FUNCTION_BLOCK basicNecessidade2Equipamentos (* Basic Function Block Type *)
  (* Standard: 61499-2 *)
  (* Version 0.0, 24/02/2026, Template *)
  PACKAGE Hidryco.HidrycoLib;
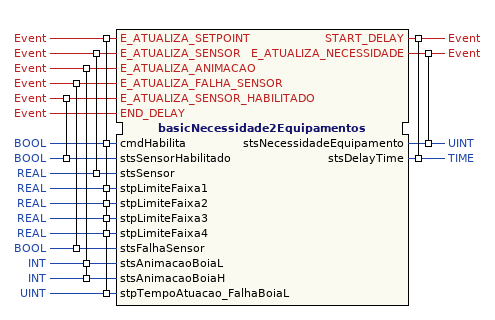
  EVENT_INPUT
    E_ATUALIZA_SETPOINT WITH stpLimiteFaixa1, stpLimiteFaixa2, stpLimiteFaixa3, stpLimiteFaixa4, stpTempoAtuacao_FalhaBoiaL, cmdHabilita;
    E_ATUALIZA_SENSOR WITH stsSensor;
    E_ATUALIZA_ANIMACAO WITH stsAnimacaoBoiaL, stsAnimacaoBoiaH;
    E_ATUALIZA_FALHA_SENSOR WITH stsFalhaSensor;
    E_ATUALIZA_SENSOR_HABILITADO WITH stsSensorHabilitado;
    END_DELAY;
  END_EVENT
  EVENT_OUTPUT
    START_DELAY WITH stsDelayTime;
    E_ATUALIZA_NECESSIDADE WITH stsNecessidadeEquipamento;
  END_EVENT
  VAR_INPUT
    cmdHabilita : BOOL;
    stsSensorHabilitado : BOOL;
    stsSensor : REAL;
    stpLimiteFaixa1 : REAL;
    stpLimiteFaixa2 : REAL;
    stpLimiteFaixa3 : REAL;
    stpLimiteFaixa4 : REAL;
    stsFalhaSensor : BOOL;
    stsAnimacaoBoiaL : INT;
    stsAnimacaoBoiaH : INT;
    stpTempoAtuacao_FalhaBoiaL : UINT; (* Tempo para equipamento ficar ligado quando bater na boia H e a boia L estiver em falha *)
  END_VAR
  VAR_OUTPUT
    stsNecessidadeEquipamento : UINT;
    stsDelayTime : TIME;
  END_VAR
  VAR
    auxiliar : INT := 0;
  END_VAR
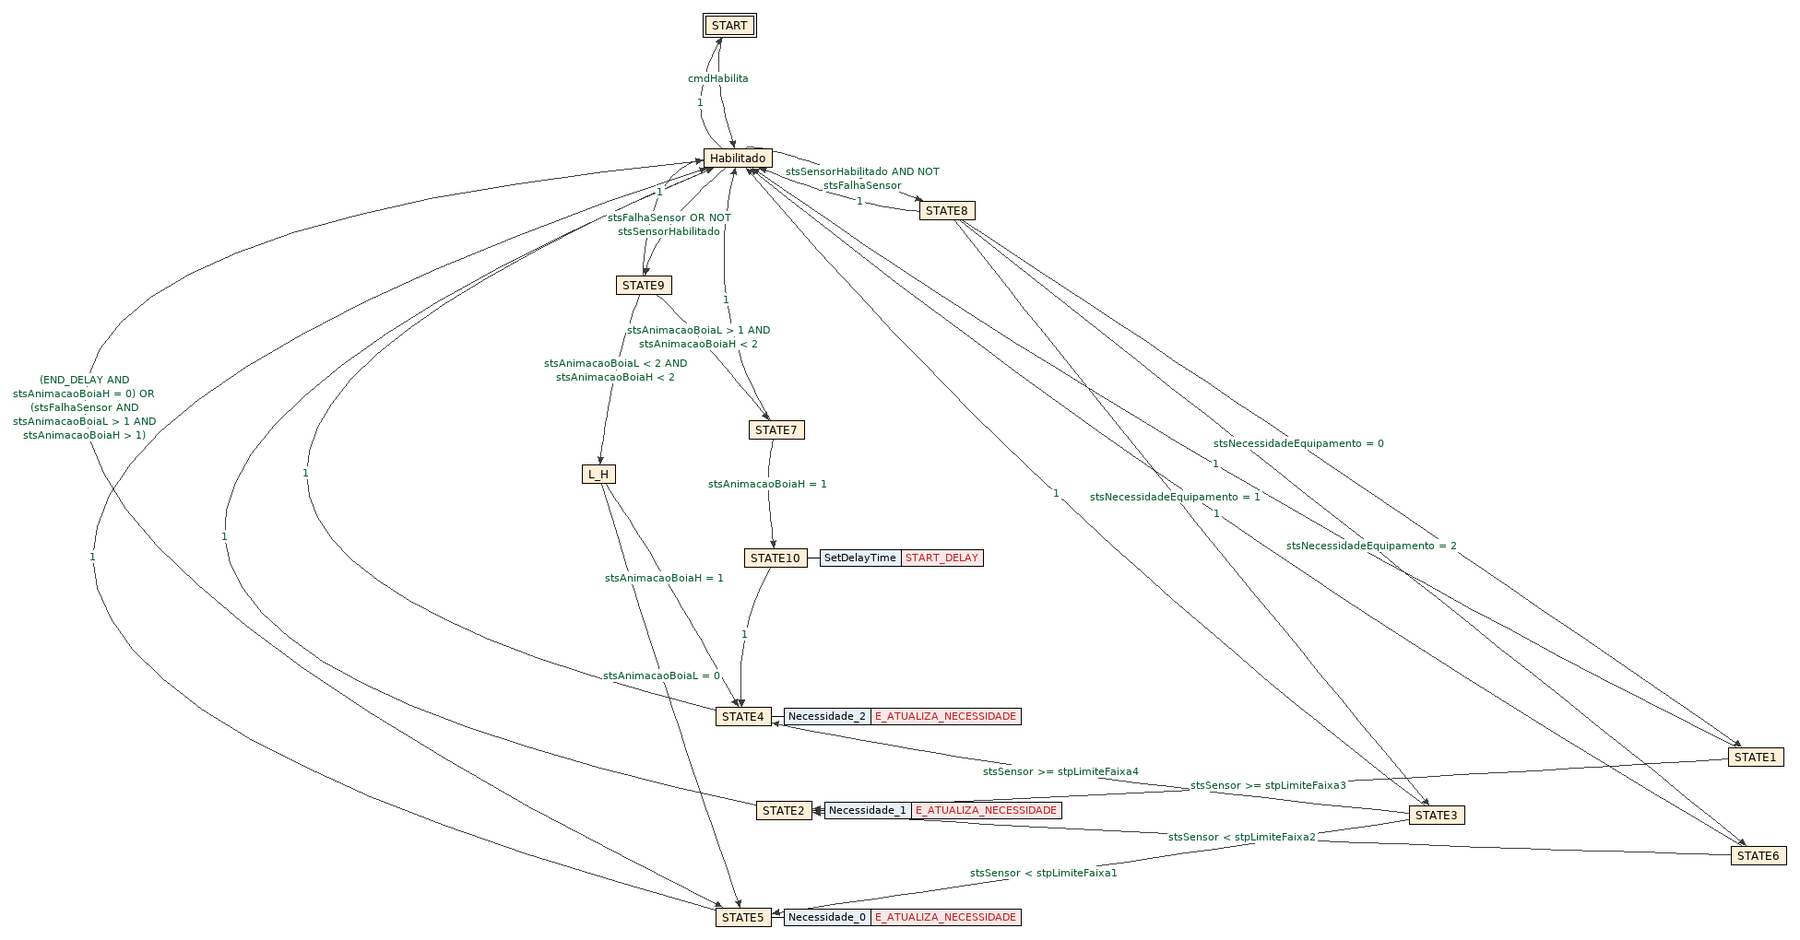
  EC_STATES
    START; (* Initial State *)
    STATE1;
    STATE2 : Necessidade_1 -> E_ATUALIZA_NECESSIDADE;
    STATE3;
    STATE4 : Necessidade_2 -> E_ATUALIZA_NECESSIDADE;
    STATE5 : Necessidade_0 -> E_ATUALIZA_NECESSIDADE;
    STATE6;
    STATE8;
    STATE9;
    L_H;
    STATE7;
    STATE10 : SetDelayTime -> START_DELAY;
    Habilitado;
  END_STATES
  EC_TRANSITIONS
    START TO Habilitado := cmdHabilita;
    Habilitado TO STATE8 := stsSensorHabilitado AND NOT stsFalhaSensor;
    STATE8 TO STATE1 := stsNecessidadeEquipamento = 0;
    STATE1 TO STATE2 := stsSensor >= stpLimiteFaixa3;
    STATE8 TO STATE3 := stsNecessidadeEquipamento = 1;
    STATE3 TO STATE4 := stsSensor >= stpLimiteFaixa4;
    STATE3 TO STATE5 := stsSensor < stpLimiteFaixa1;
    STATE8 TO STATE6 := stsNecessidadeEquipamento = 2;
    STATE6 TO STATE2 := stsSensor < stpLimiteFaixa2;
    STATE8 TO Habilitado := 1;
    Habilitado TO STATE9 := stsFalhaSensor OR NOT stsSensorHabilitado;
    STATE9 TO L_H := stsAnimacaoBoiaL < 2 AND stsAnimacaoBoiaH < 2;
    L_H TO STATE4 := stsAnimacaoBoiaH = 1;
    L_H TO STATE5 := stsAnimacaoBoiaL = 0;
    STATE9 TO STATE7 := stsAnimacaoBoiaL > 1 AND stsAnimacaoBoiaH < 2;
    STATE7 TO STATE10 := stsAnimacaoBoiaH = 1;
    STATE10 TO STATE4 := 1;
    STATE9 TO Habilitado := 1;
    Habilitado TO STATE5 := (END_DELAY AND stsAnimacaoBoiaH = 0) OR (stsFalhaSensor AND stsAnimacaoBoiaL > 1 AND stsAnimacaoBoiaH > 1);
    STATE5 TO Habilitado := 1;
    STATE2 TO Habilitado := 1;
    STATE4 TO Habilitado := 1;
    STATE1 TO Habilitado := 1;
    STATE6 TO Habilitado := 1;
    STATE3 TO Habilitado := 1;
    STATE7 TO Habilitado := 1;
    Habilitado TO START := 1;
  END_TRANSITIONS
  ALGORITHM Necessidade_1 IN ST:
stsNecessidadeEquipamento := 1;
  END_ALGORITHM
  ALGORITHM Necessidade_2 IN ST:
stsNecessidadeEquipamento := 2;
;
  END_ALGORITHM
  ALGORITHM Necessidade_0 IN ST:
stsNecessidadeEquipamento := 0;
;
  END_ALGORITHM
  ALGORITHM SetDelayTime IN ST:
stsDelayTime := DINT_TO_TIME(
    UINT_TO_DINT(stpTempoAtuacao_FalhaBoiaL) * 60000
);
  END_ALGORITHM
END_FUNCTION_BLOCK
